FUNCTION_BLOCK AnalogInputBase_HMI (* Service Interface Function Block Type *)
  (* Standard: 61499-2 *)
  (* Version 1.0.1, 1/16/2024, ApplicationLibDevTeam, Schneider Electric, First Version *)
  PACKAGE SE.Nereda;
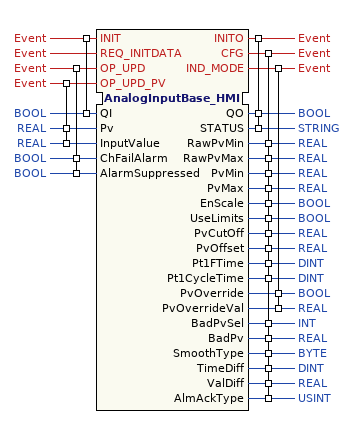
  EVENT_INPUT
    INIT WITH QI;
    REQ_INITDATA; (* Request initialization data *)
    OP_UPD WITH ChFailAlarm, AlarmSuppressed; (* Operation values update *)
    OP_UPD_PV WITH Pv, InputValue; (* Update field and processed value *)
  END_EVENT
  EVENT_OUTPUT
    INITO WITH QO, STATUS;
    CFG WITH RawPvMin, RawPvMax, PvMin, PvMax, EnScale, UseLimits, PvCutOff, PvOffset, Pt1FTime, Pt1CycleTime, BadPvSel, BadPv, SmoothType, TimeDiff, ValDiff, AlmAckType; (* Operation parameter values changed *)
    IND_MODE WITH PvOverride, PvOverrideVal; (* Indicate change in override mode and override value *)
  END_EVENT
  VAR_INPUT
    QI : BOOL;
    Pv : REAL; (* Process value *) {SET_ATTRIBUTE(Runtime.Archive.Id, 1)} {SET_ATTRIBUTE(Runtime.History.Depth, 500)} {SET_ATTRIBUTE(Runtime.History.SmoothTime, 60000)} {SET_ATTRIBUTE(Runtime.History.SmoothValue, 0.1)}
    InputValue : REAL; (* Input field value *) {SET_ATTRIBUTE(Runtime.Archive.Id, 1)} {SET_ATTRIBUTE(Runtime.History.Depth, 500)} {SET_ATTRIBUTE(Runtime.History.SmoothTime, 60000)} {SET_ATTRIBUTE(Runtime.History.SmoothValue, 0.1)}
    ChFailAlarm : BOOL; (* 1 = Analog input channel failure alarm is present *)
    AlarmSuppressed : BOOL; (* 1 = Alarm generation is suppressed *)
  END_VAR
  VAR_OUTPUT
    QO : BOOL; (* Event Output Qualifier *)
    STATUS : STRING; (* Service Status *)
    RawPvMin : REAL; (* Minimum field value *)
    RawPvMax : REAL; (* Maximum field value *)
    PvMin : REAL; (* Minimum process value *)
    PvMax : REAL; (* Maximum process value *)
    EnScale : BOOL; (* 1 = Enable scaling for value from field *)
    UseLimits : BOOL; (* 1 = Enable limiting of process value *)
    PvCutOff : REAL; (* Minimum process value limit *)
    PvOffset : REAL; (* Offset value adds to Pv *)
    Pt1FTime : DINT; (* Filter time for pt1 filter , 0.0 disables the filter functionality *)
    Pt1CycleTime : DINT; (* Cycle time of the PT1 filter in milliseconds *)
    PvOverride : BOOL; (* 1 = Override value will be considered *)
    PvOverrideVal : REAL; (* Scaled value that overrides the input value in override mode *)
    BadPvSel : INT; (* Select pv in case of bad signal (0- use input value; 1- use bad pv; 2- use last good value) *)
    BadPv : REAL; (* Process value when the signal is bad *)
    SmoothType : BYTE; (* Process value smoothing type 0=none, 1=old new, 2=value difference, 3=time difference, 4=time or value difference, 5=time and value difference *)
    TimeDiff : DINT; (* Time difference configuration  for process value smoothing *)
    ValDiff : REAL; (* Value difference configuration  for process value smoothing *)
    AlmAckType : USINT; (* 0 = not ackable; 1 = ack deletes; 2 = came has to be acked; 3 = came and gone have to be acked; 4 = pair has to be acked *)
  END_VAR
  SERVICE /
    SEQUENCE 
    END_SEQUENCE
  END_SERVICE
END_FUNCTION_BLOCK
